LIN {X 0,Y 263.568,Z 747.619,A -85,B 0,C 180,E1 823.789,E2 823.789} C_VEL
LIN {X 0,Y 270.238,Z 750.305,A -85,B 0,C 180,E1 820.195,E2 820.195} C_VEL
LIN {X 0,Y 274.458,Z 751.78,A -85,B 0,C 180,E1 817.719,E2 817.719} C_VEL
LIN {X 0,Y 276.955,Z 753.121,A -85,B 0,C 180,E1 814.763,E2 814.763} C_VEL
LIN {X 0,Y 278.461,Z 753.813,A -85,B 0,C 180,E1 812.058,E2 812.058} C_VEL
LIN {X 0,Y 278.848,Z 753.996,A -85,B 0,C 180,E1 809.589,E2 809.589} C_VEL
LIN {X 0,Y 278.04,Z 753.673,A -85,B 0,C 180,E1 806.908,E2 806.908} C_VEL
LIN {X 0,Y 275.68,Z 752.498,A -85,B 0,C 180,E1 803.616,E2 803.616} C_VEL
LIN {X 0,Y 273.788,Z 751.518,A -85,B 0,C 180,E1 801.773,E2 801.773} C_VEL
LIN {X 0,Y 266.708,Z 748.995,A -85,B 0,C 180,E1 797.883,E2 797.883} C_VEL
LIN {X 0,Y 262.237,Z 747.179,A -85,B 0,C 180,E1 795.652,E2 795.652} C_VEL
LIN {X 0,Y 252.726,Z 743.838,A -85,B 0,C 180,E1 791.722,E2 791.722} C_VEL
LIN {X 0,Y 241.319,Z 740.195,A -85,B 0,C 180,E1 787.517,E2 787.517} C_VEL
LIN {X 0,Y 229.005,Z 736.394,A -85,B 0,C 180,E1 782.963,E2 782.963} C_VEL
LIN {X 0,Y 217.311,Z 732.811,A -85,B 0,C 180,E1 778.345,E2 778.345} C_VEL
LIN {X 0,Y 213.425,Z 731.637,A -85,B 0,C 180,E1 776.725,E2 776.725} C_VEL
LIN {X 0,Y 198.051,Z 740.374,A -85,B 0,C 180,E1 781.344,E2 781.344} C_VEL
LIN {X 0,Y 188.599,Z 745.079,A -85,B 0,C 180,E1 784.811,E2 784.811} C_VEL
LIN {X 0,Y 185.006,Z 747.126,A -85,B 0,C 180,E1 786.833,E2 786.833} C_VEL
LIN {X 0,Y 179.935,Z 751.57,A -85,B 0,C 180,E1 792.976,E2 792.976} C_VEL
LIN {X 0,Y 177.39,Z 752.768,A -85,B 0,C 180,E1 795.105,E2 795.105} C_VEL
LIN {X 0,Y 168.22,Z 755.529,A -85,B 0,C 180,E1 802.144,E2 802.144} C_VEL
LIN {X 0,Y 161.989,Z 756.591,A -85,B 0,C 180,E1 810,E2 810} C_VEL
LIN {X 0,Y 168.223,Z 755.528,A -85,B 0,C 180,E1 817.856,E2 817.856} C_VEL
LIN {X 0,Y 177.571,Z 752.708,A -85,B 0,C 180,E1 825.01,E2 825.01} C_VEL
LIN {X 0,Y 190.003,Z 747.723,A -85,B 0,C 180,E1 831.612,E2 831.612} C_VEL
LIN {X 0,Y 202.682,Z 741.533,A -85,B 0,C 180,E1 836.671,E2 836.671} C_VEL
LIN {X 0,Y 212.691,Z 736.107,A -85,B 0,C 180,E1 839.884,E2 839.884} C_VEL
LIN {X 0,Y 226.557,Z 740.003,A -85,B 0,C 180,E1 834.507,E2 834.507} C_VEL
LIN {X 0,Y 237.859,Z 743.238,A -85,B 0,C 180,E1 830.376,E2 830.376} C_VEL
LIN {X 0,Y 247.484,Z 746.053,A -85,B 0,C 180,E1 826.757,E2 826.757} C_VEL
LIN {X 0,Y 256.835,Z 749.012,A -85,B 0,C 180,E1 822.819,E2 822.819} C_VEL
LIN {X 0,Y 264.414,Z 751.63,A -85,B 0,C 180,E1 818.699,E2 818.699} C_VEL
LIN {X 0,Y 266.692,Z 752.297,A -85,B 0,C 180,E1 817.323,E2 817.323} C_VEL
LIN {X 0,Y 269.382,Z 753.576,A -85,B 0,C 180,E1 814.044,E2 814.044} C_VEL
LIN {X 0,Y 270.652,Z 754.055,A -85,B 0,C 180,E1 811.482,E2 811.482} C_VEL
LIN {X 0,Y 270.803,Z 754.123,A -85,B 0,C 180,E1 809.154,E2 809.154} C_VEL
LIN {X 0,Y 269.686,Z 753.713,A -85,B 0,C 180,E1 806.387,E2 806.387} C_VEL
LIN {X 0,Y 266.98,Z 752.447,A -85,B 0,C 180,E1 802.967,E2 802.967} C_VEL
LIN {X 0,Y 265.251,Z 751.851,A -85,B 0,C 180,E1 801.766,E2 801.766} C_VEL
LIN {X 0,Y 258.231,Z 749.54,A -85,B 0,C 180,E1 797.933,E2 797.933} C_VEL
LIN {X 0,Y 255.084,Z 748.427,A -85,B 0,C 180,E1 796.399,E2 796.399} C_VEL
LIN {X 0,Y 245.508,Z 745.41,A -85,B 0,C 180,E1 792.462,E2 792.462} C_VEL
LIN {X 0,Y 234.457,Z 742.233,A -85,B 0,C 180,E1 788.39,E2 788.39} C_VEL
LIN {X 0,Y 221.891,Z 738.734,A -85,B 0,C 180,E1 783.733,E2 783.733} C_VEL
LIN {X 0,Y 212.572,Z 736.11,A -85,B 0,C 180,E1 780.097,E2 780.097} C_VEL
LIN {X 0,Y 198.289,Z 743.841,A -85,B 0,C 180,E1 784.943,E2 784.943} C_VEL
LIN {X 0,Y 185.06,Z 749.817,A -85,B 0,C 180,E1 790.759,E2 790.759} C_VEL
LIN {X 0,Y 177.39,Z 752.768,A -85,B 0,C 180,E1 795.105,E2 795.105} C_VEL
LIN {X 0,Y 174.976,Z 753.884,A -85,B 0,C 180,E1 797.481,E2 797.481} C_VEL
LIN {X 0,Y 173.588,Z 755.845,A -85,B 0,C 180,E1 804.427,E2 804.427} C_VEL
LIN {X 0,Y 172.476,Z 756.116,A -85,B 0,C 180,E1 806.6,E2 806.6} C_VEL
LIN {X 0,Y 170.137,Z 756.413,A -85,B 0,C 180,E1 810,E2 810} C_VEL
LIN {X 0,Y 176.323,Z 755.348,A -85,B 0,C 180,E1 817.493,E2 817.493} C_VEL
LIN {X 0,Y 185.485,Z 752.529,A -85,B 0,C 180,E1 824.355,E2 824.355} C_VEL
LIN {X 0,Y 197.628,Z 747.546,A -85,B 0,C 180,E1 830.739,E2 830.739} C_VEL
LIN {X 0,Y 210.013,Z 741.355,A -85,B 0,C 180,E1 835.671,E2 835.671} C_VEL
LIN {X 0,Y 212.327,Z 740.236,A -85,B 0,C 180,E1 836.372,E2 836.372} C_VEL
LIN {X 0,Y 222.807,Z 742.951,A -85,B 0,C 180,E1 832.412,E2 832.412} C_VEL
LIN {X 0,Y 231.862,Z 745.193,A -85,B 0,C 180,E1 829.129,E2 829.129} C_VEL
LIN {X 0,Y 240.445,Z 747.46,A -85,B 0,C 180,E1 825.928,E2 825.928} C_VEL
LIN {X 0,Y 249.531,Z 750.008,A -85,B 0,C 180,E1 822.115,E2 822.115} C_VEL
LIN {X 0,Y 256.633,Z 752.179,A -85,B 0,C 180,E1 818.257,E2 818.257} C_VEL
LIN {X 0,Y 258.966,Z 752.829,A -85,B 0,C 180,E1 816.873,E2 816.873} C_VEL
LIN {X 0,Y 261.665,Z 753.962,A -85,B 0,C 180,E1 813.505,E2 813.505} C_VEL
LIN {X 0,Y 262.803,Z 754.322,A -85,B 0,C 180,E1 810.654,E2 810.654} C_VEL
LIN {X 0,Y 262.562,Z 754.208,A -85,B 0,C 180,E1 808.254,E2 808.254} C_VEL
LIN {X 0,Y 261.048,Z 753.688,A -85,B 0,C 180,E1 805.607,E2 805.607} C_VEL
LIN {X 0,Y 258.705,Z 752.715,A -85,B 0,C 180,E1 802.897,E2 802.897} C_VEL
LIN {X 0,Y 252.076,Z 750.855,A -85,B 0,C 180,E1 799.257,E2 799.257} C_VEL
LIN {X 0,Y 247.962,Z 749.603,A -85,B 0,C 180,E1 797.188,E2 797.188} C_VEL
LIN {X 0,Y 238.876,Z 747.048,A -85,B 0,C 180,E1 793.447,E2 793.447} C_VEL
LIN {X 0,Y 227.636,Z 744.127,A -85,B 0,C 180,E1 789.326,E2 789.326} C_VEL
LIN {X 0,Y 215.447,Z 741.01,A -85,B 0,C 180,E1 784.823,E2 784.823} C_VEL
LIN {X 0,Y 212.087,Z 740.253,A -85,B 0,C 180,E1 783.607,E2 783.607} C_VEL
LIN {X 0,Y 199.871,Z 746.46,A -85,B 0,C 180,E1 788.275,E2 788.275} C_VEL
LIN {X 0,Y 187.815,Z 751.644,A -85,B 0,C 180,E1 794.248,E2 794.248} C_VEL
LIN {X 0,Y 178.08,Z 754.897,A -85,B 0,C 180,E1 800.956,E2 800.956} C_VEL
LIN {X 0,Y 172.476,Z 756.116,A -85,B 0,C 180,E1 806.6,E2 806.6} C_VEL
LIN {X 0,Y 172.398,Z 756.24,A -85,B 0,C 180,E1 808.049,E2 808.049} C_VEL
LIN {X 0,Y 174.875,Z 756.307,A -85,B 0,C 180,E1 810.108,E2 810.108} C_VEL
LIN {X 0,Y 180.054,Z 755.987,A -85,B 0,C 180,E1 812.935,E2 812.935} C_VEL
LIN {X 0,Y 181.149,Z 755.874,A -85,B 0,C 180,E1 813.858,E2 813.858} C_VEL
LIN {X 0,Y 189.196,Z 753.792,A -85,B 0,C 180,E1 820.966,E2 820.966} C_VEL
LIN {X 0,Y 199.071,Z 750.097,A -85,B 0,C 180,E1 826.935,E2 826.935} C_VEL
LIN {X 0,Y 209.736,Z 745.179,A -85,B 0,C 180,E1 831.827,E2 831.827} C_VEL
LIN {X 0,Y 212.328,Z 743.959,A -85,B 0,C 180,E1 832.823,E2 832.823} C_VEL
LIN {X 0,Y 225.203,Z 746.914,A -85,B 0,C 180,E1 828.105,E2 828.105} C_VEL
LIN {X 0,Y 233.883,Z 748.909,A -85,B 0,C 180,E1 824.861,E2 824.861} C_VEL
LIN {X 0,Y 242.63,Z 751.067,A -85,B 0,C 180,E1 821.167,E2 821.167} C_VEL
LIN {X 0,Y 250.076,Z 753.027,A -85,B 0,C 180,E1 817.119,E2 817.119} C_VEL
LIN {X 0,Y 251.689,Z 753.465,A -85,B 0,C 180,E1 815.928,E2 815.928} C_VEL
LIN {X 0,Y 254.074,Z 754.297,A -85,B 0,C 180,E1 812.706,E2 812.706} C_VEL
LIN {X 0,Y 254.89,Z 754.561,A -85,B 0,C 180,E1 810,E2 810} C_VEL
LIN {X 0,Y 254.211,Z 754.319,A -85,B 0,C 180,E1 807.518,E2 807.518} C_VEL
LIN {X 0,Y 251.891,Z 753.532,A -85,B 0,C 180,E1 804.306,E2 804.306} C_VEL
LIN {X 0,Y 250.518,Z 753.138,A -85,B 0,C 180,E1 803.124,E2 803.124} C_VEL
LIN {X 0,Y 243.12,Z 751.224,A -85,B 0,C 180,E1 799.096,E2 799.096} C_VEL
LIN {X 0,Y 239.473,Z 750.3,A -85,B 0,C 180,E1 797.462,E2 797.462} C_VEL
LIN {X 0,Y 231.494,Z 748.314,A -85,B 0,C 180,E1 794.212,E2 794.212} C_VEL
LIN {X 0,Y 221.256,Z 745.966,A -85,B 0,C 180,E1 790.466,E2 790.466} C_VEL
LIN {X 0,Y 212.183,Z 743.997,A -85,B 0,C 180,E1 787.198,E2 787.198} C_VEL
LIN {X 0,Y 200.07,Z 749.676,A -85,B 0,C 180,E1 792.553,E2 792.553} C_VEL
LIN {X 0,Y 189.598,Z 753.665,A -85,B 0,C 180,E1 798.749,E2 798.749} C_VEL
LIN {X 0,Y 181.37,Z 755.846,A -85,B 0,C 180,E1 805.891,E2 805.891} C_VEL
LIN {X 0,Y 178.286,Z 756.235,A -85,B 0,C 180,E1 810,E2 810} C_VEL
LIN {X 0,Y 181.149,Z 755.874,A -85,B 0,C 180,E1 813.858,E2 813.858} C_VEL
LIN {X 0,Y 184.313,Z 755.487,A -85,B 0,C 180,E1 816.079,E2 816.079} C_VEL
LIN {X 0,Y 197.269,Z 753.379,A -85,B 0,C 180,E1 821.104,E2 821.104} C_VEL
LIN {X 0,Y 200.621,Z 752.445,A -85,B 0,C 180,E1 822.742,E2 822.742} C_VEL
LIN {X 0,Y 211.426,Z 747.914,A -85,B 0,C 180,E1 828.471,E2 828.471} C_VEL
LIN {X 0,Y 212.878,Z 747.332,A -85,B 0,C 180,E1 829.043,E2 829.043} C_VEL
LIN {X 0,Y 220.387,Z 748.785,A -85,B 0,C 180,E1 826.335,E2 826.335} C_VEL
LIN {X 0,Y 227.451,Z 750.255,A -85,B 0,C 180,E1 823.704,E2 823.704} C_VEL
LIN {X 0,Y 235.096,Z 751.867,A -85,B 0,C 180,E1 820.536,E2 820.536} C_VEL
LIN {X 0,Y 242.745,Z 753.576,A -85,B 0,C 180,E1 816.385,E2 816.385} C_VEL
LIN {X 0,Y 244.181,Z 753.917,A -85,B 0,C 180,E1 815.168,E2 815.168} C_VEL
LIN {X 0,Y 246.214,Z 754.518,A -85,B 0,C 180,E1 812.327,E2 812.327} C_VEL
LIN {X 0,Y 246.866,Z 754.719,A -85,B 0,C 180,E1 809.768,E2 809.768} C_VEL
LIN {X 0,Y 245.974,Z 754.472,A -85,B 0,C 180,E1 807.204,E2 807.204} C_VEL
LIN {X 0,Y 243.335,Z 753.672,A -85,B 0,C 180,E1 803.939,E2 803.939} C_VEL
LIN {X 0,Y 235.596,Z 751.998,A -85,B 0,C 180,E1 799.734,E2 799.734} C_VEL
LIN {X 0,Y 228.097,Z 750.39,A -85,B 0,C 180,E1 796.568,E2 796.568} C_VEL
LIN {X 0,Y 222.975,Z 749.323,A -85,B 0,C 180,E1 794.608,E2 794.608} C_VEL
LIN {X 0,Y 214.161,Z 747.567,A -85,B 0,C 180,E1 791.403,E2 791.403} C_VEL
LIN {X 0,Y 212.669,Z 747.36,A -85,B 0,C 180,E1 790.966,E2 790.966} C_VEL
LIN {X 0,Y 201.224,Z 752.229,A -85,B 0,C 180,E1 796.89,E2 796.89} C_VEL
LIN {X 0,Y 192.543,Z 754.989,A -85,B 0,C 180,E1 803.141,E2 803.141} C_VEL
LIN {X 0,Y 186.438,Z 756.057,A -85,B 0,C 180,E1 810,E2 810} C_VEL
LIN {X 0,Y 192.544,Z 754.989,A -85,B 0,C 180,E1 816.859,E2 816.859} C_VEL
LIN {X 0,Y 200.621,Z 752.445,A -85,B 0,C 180,E1 822.742,E2 822.742} C_VEL
LIN {X 0,Y 202.549,Z 752.106,A -85,B 0,C 180,E1 823.234,E2 823.234} C_VEL
LIN {X 0,Y 206.208,Z 751.827,A -85,B 0,C 180,E1 823.408,E2 823.408} C_VEL
LIN {X 0,Y 211.842,Z 751.713,A -85,B 0,C 180,E1 823.039,E2 823.039} C_VEL
LIN {X 0,Y 217.412,Z 751.87,A -85,B 0,C 180,E1 822.164,E2 822.164} C_VEL
LIN {X 0,Y 224.077,Z 752.307,A -85,B 0,C 180,E1 820.694,E2 820.694} C_VEL
LIN {X 0,Y 228.581,Z 752.827,A -85,B 0,C 180,E1 819.24,E2 819.24} C_VEL
LIN {X 0,Y 229.829,Z 753.049,A -85,B 0,C 180,E1 818.655,E2 818.655} C_VEL
LIN {X 0,Y 235.963,Z 754.129,A -85,B 0,C 180,E1 815.245,E2 815.245} C_VEL
LIN {X 0,Y 238.243,Z 754.716,A -85,B 0,C 180,E1 812.164,E2 812.164} C_VEL
LIN {X 0,Y 238.865,Z 754.894,A -85,B 0,C 180,E1 809.76,E2 809.76} C_VEL
LIN {X 0,Y 237.979,Z 754.674,A -85,B 0,C 180,E1 807.351,E2 807.351} C_VEL
LIN {X 0,Y 235.684,Z 754.069,A -85,B 0,C 180,E1 804.523,E2 804.523} C_VEL
LIN {X 0,Y 228.606,Z 752.789,A -85,B 0,C 180,E1 800.688,E2 800.688} C_VEL
LIN {X 0,Y 222.406,Z 751.692,A -85,B 0,C 180,E1 798.066,E2 798.066} C_VEL
LIN {X 0,Y 217.352,Z 750.757,A -85,B 0,C 180,E1 796.089,E2 796.089} C_VEL
LIN {X 0,Y 213.828,Z 750.165,A -85,B 0,C 180,E1 794.822,E2 794.822} C_VEL
LIN {X 0,Y 204.145,Z 753.813,A -85,B 0,C 180,E1 800.7,E2 800.7} C_VEL
LIN {X 0,Y 196.874,Z 755.593,A -85,B 0,C 180,E1 807.089,E2 807.089} C_VEL
LIN {X 0,Y 194.592,Z 755.879,A -85,B 0,C 180,E1 810,E2 810} C_VEL
LIN {X 0,Y 200.663,Z 754.809,A -85,B 0,C 180,E1 816.58,E2 816.58} C_VEL
LIN {X 0,Y 209.347,Z 751.987,A -85,B 0,C 180,E1 822.69,E2 822.69} C_VEL
LIN {X 0,Y 213.841,Z 750.165,A -85,B 0,C 180,E1 825.178,E2 825.178} C_VEL
LIN {X 0,Y 220.929,Z 751.39,A -85,B 0,C 180,E1 822.545,E2 822.545} C_VEL
LIN {X 0,Y 228.144,Z 752.692,A -85,B 0,C 180,E1 819.56,E2 819.56} C_VEL
LIN {X 0,Y 229.829,Z 753.049,A -85,B 0,C 180,E1 818.655,E2 818.655} C_VEL
LIN {X 0,Y 230.987,Z 753.589,A -85,B 0,C 180,E1 817.418,E2 817.418} C_VEL
LIN {X 0,Y 230.466,Z 754.219,A -85,B 0,C 180,E1 815.564,E2 815.564} C_VEL
LIN {X 0,Y 229.602,Z 754.805,A -85,B 0,C 180,E1 813.26,E2 813.26} C_VEL
LIN {X 0,Y 229.833,Z 754.856,A -85,B 0,C 180,E1 812.686,E2 812.686} C_VEL
LIN {X 0,Y 230.856,Z 755.069,A -85,B 0,C 180,E1 810.248,E2 810.248} C_VEL
LIN {X 0,Y 230.291,Z 754.913,A -85,B 0,C 180,E1 808.01,E2 808.01} C_VEL
LIN {X 0,Y 228.201,Z 754.485,A -85,B 0,C 180,E1 805.225,E2 805.225} C_VEL
LIN {X 0,Y 221.146,Z 753.433,A -85,B 0,C 180,E1 801.42,E2 801.42} C_VEL
LIN {X 0,Y 215.283,Z 752.584,A -85,B 0,C 180,E1 799.024,E2 799.024} C_VEL
LIN {X 0,Y 207.544,Z 754.941,A -85,B 0,C 180,E1 804.749,E2 804.749} C_VEL
LIN {X 0,Y 202.748,Z 755.7,A -85,B 0,C 180,E1 810,E2 810} C_VEL
LIN {X 0,Y 208.787,Z 754.629,A -85,B 0,C 180,E1 816.323,E2 816.323} C_VEL
LIN {X 0,Y 215.322,Z 752.583,A -85,B 0,C 180,E1 820.974,E2 820.974} C_VEL
LIN {X 0,Y 221.382,Z 753.481,A -85,B 0,C 180,E1 818.454,E2 818.454} C_VEL
LIN {X 0,Y 228.196,Z 754.485,A -85,B 0,C 180,E1 814.775,E2 814.775} C_VEL
LIN {X 0,Y 229.833,Z 754.856,A -85,B 0,C 180,E1 812.686,E2 812.686} C_VEL
LIN {X 0,Y 229.621,Z 754.984,A -85,B 0,C 180,E1 811.6,E2 811.6} C_VEL
LIN {X 0,Y 227.095,Z 755.168,A -85,B 0,C 180,E1 810.043,E2 810.043} C_VEL
LIN {X 0,Y 222.071,Z 755.066,A -85,B 0,C 180,E1 807.556,E2 807.556} C_VEL
LIN {X 0,Y 221.456,Z 755.012,A -85,B 0,C 180,E1 806.972,E2 806.972} C_VEL
LIN {X 0,Y 220.011,Z 754.809,A -85,B 0,C 180,E1 805.57,E2 805.57} C_VEL
LIN {X 0,Y 216.916,Z 754.449,A -85,B 0,C 180,E1 803.915,E2 803.915} C_VEL
LIN {X 0,Y 210.906,Z 755.522,A -85,B 0,C 180,E1 810,E2 810} C_VEL
LIN {X 0,Y 216.933,Z 754.448,A -85,B 0,C 180,E1 816.085,E2 816.085} C_VEL
LIN {X 0,Y 220.757,Z 754.93,A -85,B 0,C 180,E1 813.895,E2 813.895} C_VEL
LIN {X 0,Y 222.651,Z 755.176,A -85,B 0,C 180,E1 811.029,E2 811.029} C_VEL
LIN {X 0,Y 222.768,Z 755.197,A -85,B 0,C 180,E1 809.229,E2 809.229} C_VEL
LIN {X 0,Y 221.456,Z 755.012,A -85,B 0,C 180,E1 806.972,E2 806.972} C_VEL
LIN {X 0,Y 221.069,Z 757.012,A -85,B 0,C 180,E1 806.452,E2 806.452} C_VEL
LIN {X 0,Y 221.069,Z 783.5,A -85,B 0,C 180,E1 806.452,E2 806.452} C_VEL
LIN {X 0,Y 221.069,Z 783.5,A -85,B 0,C 180,E1 806.452,E2 806.452}

QRS_NEXT_CUT()

QRS_NEXT()
QRS_HOME()

END
